Yaskawa INFORM job: profile_long_22-06-23_planes_program.JBI

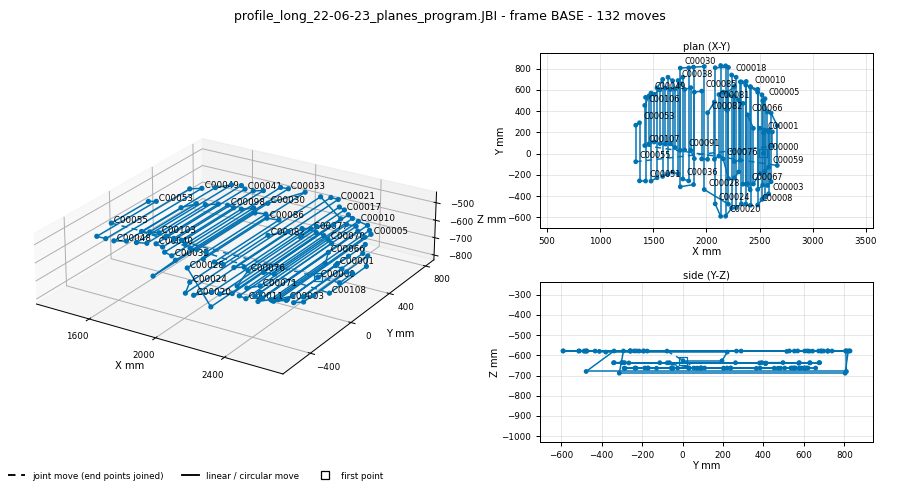
[picture p0: tool path of profile_long_22-06-23_planes_program.JBI in frame BASE, 132 of 138 moves have a stored position in this frame; points joined in program order, loops and branches not executed]
/JOB
//NAME profile_long_22-06-23_planes_program
//POS
///NPOS 132,0,132,0,0,0
///TOOL 0
///POSTYPE BASE
///RECTAN
///RCONF 0,0,0,0,0,0,0,0,0,0,0,0,0,0,0,0,0,0,0,0,0,0,0,0
C00000=2536.598527,2.004229,-626.796948,180.000000,-40.759430,5.000000
C00001=2536.598527,195.381529,-626.796948,180.000000,-40.759430,5.000000
C00002=2584.876284,221.287942,-584.317365,-175.000000,-13.943179,-5.000000
C00003=2584.876284,-379.409058,-584.317365,-175.000000,-13.943179,-5.000000
C00004=2551.646255,-411.098731,-580.824727,-175.000000,-9.046207,-5.000000
C00005=2551.646255,515.775269,-580.824727,-175.000000,-9.046207,-5.000000
C00006=2522.447995,553.060580,-579.157659,-175.000000,-5.000000,-5.000000
C00007=2522.447995,-431.960420,-579.157659,-175.000000,-5.000000,-5.000000
C00008=2482.537570,-484.099297,-578.765660,-175.000000,-5.000000,-5.000000
C00009=2482.537570,604.222703,-578.765660,-175.000000,-5.000000,-5.000000
C00010=2415.297292,626.844339,-579.595482,-175.000000,-5.093670,-5.000000
C00011=2415.297292,-486.433661,-579.595482,-175.000000,-5.093670,-5.000000
C00012=2371.138050,-475.933835,-579.494357,-174.708222,-5.000000,-5.000000
C00013=2371.138050,643.093165,-579.494357,-174.708222,-5.000000,-5.000000
C00014=2329.401999,672.992910,-578.789014,-175.000000,-5.000000,-5.000000
C00015=2329.401999,-473.773090,-578.789014,-175.000000,-5.000000,-5.000000
C00016=2279.866175,-509.701478,-578.799632,-175.000000,-5.000000,-5.000000
C00017=2279.866175,718.157522,-578.799632,-175.000000,-5.000000,-5.000000
C00018=2237.397039,739.175601,-578.936011,-175.000000,5.000000,5.000000
C00019=2237.397039,-513.272399,-578.936011,-175.000000,5.000000,5.000000
C00020=2181.203851,-589.383224,-578.612215,-175.000000,-5.000000,-5.000000
C00021=2181.203851,825.471776,-578.612215,-175.000000,-5.000000,-5.000000
C00022=2134.330586,828.239527,-578.541326,-175.000000,5.000000,5.000000
C00023=2134.330586,-591.013473,-578.541326,-175.000000,5.000000,5.000000
C00024=2082.887251,-473.418612,-578.562736,-175.000000,-5.000000,-5.000000
C00025=2082.887251,807.537388,-578.562736,-175.000000,-5.000000,-5.000000
C00026=2207.274470,810.333102,-680.036930,180.000000,-60.576725,-175.000000
C00027=2207.274470,-476.558898,-680.036930,180.000000,-60.576725,-175.000000
C00028=1979.808747,-338.711878,-578.882836,175.000000,-5.000000,5.000000
C00029=1979.808747,819.410122,-578.882836,175.000000,-5.000000,5.000000
C00030=1754.548583,804.064826,-688.690980,-180.000000,-63.385371,5.000000
C00031=1754.548583,-312.497174,-688.690980,-180.000000,-63.385371,5.000000
C00032=1878.672623,-292.005936,-578.782354,-175.000000,-5.000000,-5.000000
C00033=1878.672623,813.221064,-578.782354,-175.000000,-5.000000,-5.000000
C00034=1833.476054,806.462778,-578.669752,-175.000000,5.000000,5.000000
C00035=1833.476054,-257.597222,-578.669752,-175.000000,5.000000,5.000000
C00036=1778.042267,-239.268025,-578.589561,-175.000000,-5.000000,-5.000000
C00037=1778.042267,718.215975,-578.589561,-175.000000,-5.000000,-5.000000
C00038=1733.644709,686.648138,-578.598733,-175.000000,5.000000,5.000000
C00039=1733.644709,-191.224862,-578.598733,-175.000000,5.000000,5.000000
C00040=1681.906052,-174.446903,-579.093313,-174.869317,-5.000000,-5.000000
C00041=1681.906052,685.490097,-579.093313,-174.869317,-5.000000,-5.000000
C00042=1638.342652,718.026100,-579.226961,-174.651796,5.000000,5.000000
C00043=1638.342652,-193.738900,-579.226961,-174.651796,5.000000,5.000000
C00044=1588.489893,-215.075375,-578.912946,-175.000000,5.000000,5.000000
C00045=1588.489893,697.558625,-578.912946,-175.000000,5.000000,5.000000
C00046=1535.192030,617.546074,-578.595892,-175.000000,5.000000,5.000000
C00047=1535.192030,-227.909926,-578.595892,-175.000000,5.000000,5.000000
C00048=1479.024488,-259.321700,-578.487796,-175.000000,-5.000000,-5.000000
C00049=1479.024488,569.507300,-578.487796,-175.000000,-5.000000,-5.000000
C00050=1427.681228,528.296448,-578.498191,-175.000000,-5.000000,-5.000000
C00051=1427.681228,-258.567552,-578.498191,-175.000000,-5.000000,-5.000000
C00052=1370.509818,-257.169723,-579.196862,-175.000000,-5.000000,-5.000000
C00053=1370.509818,289.799277,-579.196862,-175.000000,-5.000000,-5.000000
C00054=1335.137114,266.870471,-579.315076,-174.222618,5.000000,5.000000
C00055=1335.137114,-76.747119,-579.315076,-174.222618,5.000000,5.000000
C00056=2620.892174,69.597499,-663.927425,-175.000000,-5.970680,-5.000000
C00057=2620.892174,203.269499,-663.927425,-175.000000,-5.970680,-5.000000
C00058=2586.719126,203.219520,-664.058983,-175.000000,-6.519691,-5.000000
C00059=2586.719126,-128.491880,-664.058983,-175.000000,-6.519691,-5.000000
C00060=2549.218062,-169.186736,-663.035875,-175.000000,-5.000000,-5.000000
C00061=2549.218062,220.267264,-663.035875,-175.000000,-5.000000,-5.000000
C00062=2501.928648,238.510728,-662.934382,-175.000000,-5.000000,-5.000000
C00063=2501.928648,-186.315272,-662.934382,-175.000000,-5.000000,-5.000000
C00064=2442.218519,-286.118849,-663.619592,-175.000000,-5.000000,-5.000000
C00065=2442.218519,237.348151,-663.619592,-175.000000,-5.000000,-5.000000
C00066=2386.975534,364.986863,-664.629836,-175.000000,-6.426249,-5.000000
C00067=2386.975534,-284.554137,-664.629836,-175.000000,-6.426249,-5.000000
C00068=2344.656271,-288.375145,-664.175751,-174.334966,-5.000000,-5.000000
C00069=2344.656271,472.281855,-664.175751,-174.334966,-5.000000,-5.000000
C00070=2304.131653,505.389159,-663.311980,-175.000000,-5.000000,-5.000000
C00071=2304.131653,-172.640841,-663.311980,-175.000000,-5.000000,-5.000000
C00072=2261.601953,-229.577589,-663.108050,-175.000000,5.000000,5.000000
C00073=2261.601953,535.571411,-663.108050,-175.000000,5.000000,5.000000
C00074=2207.631703,549.091120,-663.094418,-175.000000,-5.000000,-5.000000
C00075=2207.631703,-235.056880,-663.094418,-175.000000,-5.000000,-5.000000
C00076=2157.705907,-50.195973,-663.190262,-175.000000,-5.000000,-5.000000
C00077=2157.705907,578.112227,-663.190262,-175.000000,-5.000000,-5.000000
C00078=2117.384571,554.964059,-663.272967,-175.000000,5.000000,5.000000
C00079=2117.384571,-24.002741,-663.272967,-175.000000,5.000000,5.000000
C00080=2075.316641,-54.334376,-663.755737,-175.000000,5.000000,5.000000
C00081=2075.316641,484.592084,-663.755737,-175.000000,5.000000,5.000000
C00082=2011.362668,383.612144,-662.868334,-175.000000,5.000000,5.000000
C00083=2011.362668,-54.365046,-662.868334,-175.000000,5.000000,5.000000
C00084=1955.568168,-51.052863,-662.936976,-175.000000,-5.000000,-5.000000
C00085=1955.568168,587.650347,-662.936976,-175.000000,-5.000000,-5.000000
C00086=1886.476770,577.607332,-664.409273,-175.000000,-6.578793,-5.000000
C00087=1886.476770,-47.565468,-664.409273,-175.000000,-6.578793,-5.000000
C00088=1853.319685,30.306517,-663.161911,-175.000000,-5.000000,-5.000000
C00089=1853.319685,620.187017,-663.161911,-175.000000,-5.000000,-5.000000
C00090=1795.902904,603.212791,-663.607779,-175.000000,-5.000000,-5.000000
C00091=1795.902904,32.566791,-663.607779,-175.000000,-5.000000,-5.000000
C00092=1754.320672,29.884224,-663.128444,-175.000000,-5.000000,-5.000000
C00093=1754.320672,658.069624,-663.128444,-175.000000,-5.000000,-5.000000
C00094=1706.487707,608.289945,-663.248076,-175.000000,-5.000000,-5.000000
C00095=1706.487707,55.796945,-663.248076,-175.000000,-5.000000,-5.000000
C00096=1661.200144,91.026205,-663.280761,-175.000000,5.000000,5.000000
C00097=1661.200144,602.759205,-663.280761,-175.000000,5.000000,5.000000
C00098=1614.593748,614.772666,-663.283828,-175.000000,5.000000,5.000000
C00099=1614.593748,89.101666,-663.283828,-175.000000,5.000000,5.000000
C00100=1563.647765,93.498876,-663.173439,-175.000000,5.000000,5.000000
C00101=1563.647765,600.604876,-663.173439,-175.000000,5.000000,5.000000
C00102=1509.008634,557.173107,-663.116501,-175.000000,-5.000000,-5.000000
C00103=1509.008634,109.180107,-663.116501,-175.000000,-5.000000,-5.000000
C00104=1460.475573,92.235715,-663.137962,-175.000000,5.000000,5.000000
C00105=1460.475573,542.485715,-663.137962,-175.000000,5.000000,5.000000
C00106=1419.885939,453.285784,-663.782579,-174.716746,5.000000,5.000000
C00107=1419.885939,75.467784,-663.782579,-174.716746,5.000000,5.000000
C00108=2666.772027,-112.261769,-636.738710,-175.000000,-5.000000,-5.000000
C00109=2666.772027,261.995331,-636.738710,-175.000000,-5.000000,-5.000000
C00110=2608.951402,381.030762,-637.876475,-175.000000,-6.408807,-5.000000
C00111=2608.951402,-264.972238,-637.876475,-175.000000,-6.408807,-5.000000
C00112=2573.873265,-300.284116,-636.280803,-175.000000,-5.000000,-5.000000
C00113=2573.873265,391.651884,-636.280803,-175.000000,-5.000000,-5.000000
C00114=2530.108738,496.843725,-636.212429,-175.000000,-5.000000,-5.000000
C00115=2530.108738,-296.777275,-636.212429,-175.000000,-5.000000,-5.000000
C00116=2482.744724,-338.156662,-636.192294,-175.000000,5.000000,5.000000
C00117=2482.744724,577.032338,-636.192294,-175.000000,5.000000,5.000000
C00118=2412.197987,628.980369,-637.311364,-175.000000,-5.483082,-5.000000
C00119=2412.197987,-340.849631,-637.311364,-175.000000,-5.483082,-5.000000
C00120=2374.660605,-286.469165,-636.397181,-175.000000,-5.000000,-5.000000
C00121=2374.660605,678.109835,-636.397181,-175.000000,-5.000000,-5.000000
C00122=2319.427106,674.681551,-636.677680,-175.000000,-5.000000,-5.000000
C00123=2319.427106,-64.307929,-636.677680,-175.000000,-5.000000,-5.000000
C00124=2263.641899,-74.961593,-637.096476,-175.000000,-5.070659,-5.000000
C00125=2263.641899,630.971707,-637.096476,-175.000000,-5.070659,-5.000000
C00126=2194.360285,574.343532,-639.505887,-175.000000,-10.645317,-5.000000
C00127=2194.360285,411.097532,-639.505887,-175.000000,-10.645317,-5.000000
C00128=2194.360285,411.097532,-639.505887,-175.000000,-10.645317,-5.000000
C00129=2194.360285,411.097532,-639.505887,-175.000000,-10.645317,-5.000000
C00130=2194.360285,411.097532,-639.505887,-175.000000,-10.645317,-5.000000
C00131=2194.360285,411.097532,-639.505887,-175.000000,-10.645317,-5.000000
///POSTYPE PULSE
///PULSE
EC00000=0
EC00001=0
EC00002=0
EC00003=0
EC00004=0
EC00005=0
EC00006=0
EC00007=0
EC00008=0
EC00009=0
EC00010=0
EC00011=0
EC00012=0
EC00013=0
EC00014=0
EC00015=0
EC00016=0
EC00017=0
EC00018=0
EC00019=0
EC00020=0
EC00021=0
EC00022=0
EC00023=0
EC00024=0
EC00025=0
EC00026=0
EC00027=0
EC00028=0
EC00029=0
EC00030=0
EC00031=0
EC00032=0
EC00033=0
EC00034=0
EC00035=0
EC00036=0
EC00037=0
EC00038=0
EC00039=0
EC00040=0
EC00041=0
EC00042=0
EC00043=0
EC00044=0
EC00045=0
EC00046=0
EC00047=0
EC00048=0
EC00049=0
EC00050=0
EC00051=0
EC00052=0
EC00053=0
EC00054=0
EC00055=0
EC00056=0
EC00057=0
EC00058=0
EC00059=0
EC00060=0
EC00061=0
EC00062=0
EC00063=0
EC00064=0
EC00065=0
EC00066=0
EC00067=0
EC00068=0
EC00069=0
EC00070=0
EC00071=0
EC00072=0
EC00073=0
EC00074=0
EC00075=0
EC00076=0
EC00077=0
EC00078=0
EC00079=0
EC00080=0
EC00081=0
EC00082=0
EC00083=0
EC00084=0
EC00085=0
EC00086=0
EC00087=0
EC00088=0
EC00089=0
EC00090=0
EC00091=0
EC00092=0
EC00093=0
EC00094=0
EC00095=0
EC00096=0
EC00097=0
EC00098=0
EC00099=0
EC00100=0
EC00101=0
EC00102=0
EC00103=0
EC00104=0
EC00105=0
EC00106=0
EC00107=0
EC00108=0
EC00109=0
EC00110=0
EC00111=0
EC00112=0
EC00113=0
EC00114=0
EC00115=0
EC00116=0
EC00117=0
EC00118=0
EC00119=0
EC00120=0
EC00121=0
EC00122=0
EC00123=0
EC00124=0
EC00125=0
EC00126=0
EC00127=0
EC00128=92160
EC00129=184320
EC00130=276480
EC00131=368640
//INST
///DATE 2023/06/22 16:21
///ATTR SC,RW,RJ
////FRAME BASE
///GROUP1 RB1,ST1
NOP
MOVJ P009 EX000 VJ=15.00
MOVJ C00000 EC00000 VJ=15.0
CALL JOB:SPYON
MOVL C00001 EC00001 V=150.0
MOVL C00002 EC00002 V=150.0
MOVL C00003 EC00003 V=150.0
MOVL C00004 EC00004 V=150.0
MOVL C00005 EC00005 V=150.0
MOVL C00006 EC00006 V=150.0
MOVL C00007 EC00007 V=150.0
MOVL C00008 EC00008 V=150.0
MOVL C00009 EC00009 V=150.0
MOVL C00010 EC00010 V=150.0
MOVL C00011 EC00011 V=150.0
MOVL C00012 EC00012 V=150.0
MOVL C00013 EC00013 V=150.0
MOVL C00014 EC00014 V=150.0
MOVL C00015 EC00015 V=150.0
MOVL C00016 EC00016 V=150.0
MOVL C00017 EC00017 V=150.0
MOVL C00018 EC00018 V=150.0
MOVL C00019 EC00019 V=150.0
MOVL C00020 EC00020 V=150.0
MOVL C00021 EC00021 V=150.0
MOVL C00022 EC00022 V=150.0
MOVL C00023 EC00023 V=150.0
MOVL C00024 EC00024 V=150.0
MOVL C00025 EC00025 V=150.0
MOVL C00026 EC00026 V=150.0
MOVL C00027 EC00027 V=150.0
MOVL C00028 EC00028 V=150.0
MOVL C00029 EC00029 V=150.0
MOVL C00030 EC00030 V=150.0
MOVL C00031 EC00031 V=150.0
MOVL C00032 EC00032 V=150.0
MOVL C00033 EC00033 V=150.0
MOVL C00034 EC00034 V=150.0
MOVL C00035 EC00035 V=150.0
MOVL C00036 EC00036 V=150.0
MOVL C00037 EC00037 V=150.0
MOVL C00038 EC00038 V=150.0
MOVL C00039 EC00039 V=150.0
MOVL C00040 EC00040 V=150.0
MOVL C00041 EC00041 V=150.0
MOVL C00042 EC00042 V=150.0
MOVL C00043 EC00043 V=150.0
MOVL C00044 EC00044 V=150.0
MOVL C00045 EC00045 V=150.0
MOVL C00046 EC00046 V=150.0
MOVL C00047 EC00047 V=150.0
MOVL C00048 EC00048 V=150.0
MOVL C00049 EC00049 V=150.0
MOVL C00050 EC00050 V=150.0
MOVL C00051 EC00051 V=150.0
MOVL C00052 EC00052 V=150.0
MOVL C00053 EC00053 V=150.0
MOVL C00054 EC00054 V=150.0
MOVL C00055 EC00055 V=150.0
CALL JOB:SPYOF
MOVJ C00056 EC00056 VJ=15.0
CALL JOB:SPYON
MOVL C00057 EC00057 V=150.0
MOVL C00058 EC00058 V=150.0
MOVL C00059 EC00059 V=150.0
MOVL C00060 EC00060 V=150.0
MOVL C00061 EC00061 V=150.0
MOVL C00062 EC00062 V=150.0
MOVL C00063 EC00063 V=150.0
MOVL C00064 EC00064 V=150.0
MOVL C00065 EC00065 V=150.0
MOVL C00066 EC00066 V=150.0
MOVL C00067 EC00067 V=150.0
MOVL C00068 EC00068 V=150.0
MOVL C00069 EC00069 V=150.0
MOVL C00070 EC00070 V=150.0
MOVL C00071 EC00071 V=150.0
MOVL C00072 EC00072 V=150.0
MOVL C00073 EC00073 V=150.0
MOVL C00074 EC00074 V=150.0
MOVL C00075 EC00075 V=150.0
MOVL C00076 EC00076 V=150.0
MOVL C00077 EC00077 V=150.0
MOVL C00078 EC00078 V=150.0
MOVL C00079 EC00079 V=150.0
MOVL C00080 EC00080 V=150.0
MOVL C00081 EC00081 V=150.0
MOVL C00082 EC00082 V=150.0
MOVL C00083 EC00083 V=150.0
MOVL C00084 EC00084 V=150.0
MOVL C00085 EC00085 V=150.0
MOVL C00086 EC00086 V=150.0
MOVL C00087 EC00087 V=150.0
MOVL C00088 EC00088 V=150.0
MOVL C00089 EC00089 V=150.0
MOVL C00090 EC00090 V=150.0
MOVL C00091 EC00091 V=150.0
MOVL C00092 EC00092 V=150.0
MOVL C00093 EC00093 V=150.0
MOVL C00094 EC00094 V=150.0
MOVL C00095 EC00095 V=150.0
MOVL C00096 EC00096 V=150.0
MOVL C00097 EC00097 V=150.0
MOVL C00098 EC00098 V=150.0
MOVL C00099 EC00099 V=150.0
MOVL C00100 EC00100 V=150.0
MOVL C00101 EC00101 V=150.0
MOVL C00102 EC00102 V=150.0
MOVL C00103 EC00103 V=150.0
MOVL C00104 EC00104 V=150.0
MOVL C00105 EC00105 V=150.0
MOVL C00106 EC00106 V=150.0
MOVL C00107 EC00107 V=150.0
CALL JOB:SPYOF
MOVJ C00108 EC00108 VJ=15.0
CALL JOB:SPYON
MOVL C00109 EC00109 V=150.0
MOVL C00110 EC00110 V=150.0
MOVL C00111 EC00111 V=150.0
MOVL C00112 EC00112 V=150.0
MOVL C00113 EC00113 V=150.0
MOVL C00114 EC00114 V=150.0
MOVL C00115 EC00115 V=150.0
MOVL C00116 EC00116 V=150.0
MOVL C00117 EC00117 V=150.0
MOVL C00118 EC00118 V=150.0
MOVL C00119 EC00119 V=150.0
MOVL C00120 EC00120 V=150.0
MOVL C00121 EC00121 V=150.0
MOVL C00122 EC00122 V=150.0
MOVL C00123 EC00123 V=150.0
MOVL C00124 EC00124 V=150.0
MOVL C00125 EC00125 V=150.0
MOVL C00126 EC00126 V=150.0
MOVL C00127 EC00127 V=150.0
CALL JOB:SPYOF
MOVJ P009 VJ=15.00
MOVJ P009 VJ=15.00
MOVL C00128 EC00128 V=150.0
MOVJ P009 VJ=15.00
MOVL C00129 EC00129 V=150.0
MOVJ P009 VJ=15.00
MOVL C00130 EC00130 V=150.0
MOVJ P009 VJ=15.00
MOVL C00131 EC00131 V=150.0
END
